// TIA Portal project "FactoryIO_Template_S7-1200_V14" (V14)
// Vorlageprojekt für das Buch mit Zielsystem S7-1200

(* hardware
DEVICE "S7-1200-Station_1"  S7-1200 Station
   slot 0: "Baugruppenträger_0"  Rack  V1.0
   slot 1: "PLC_1"  CPU 1214C DC/DC/Rly  6ES7 214-1HG40-0XB0  V4.2
   slot 3: "DQ 4x24VDC_1"  DQ4 signal board (200 kHz)  6ES7 222-1BD30-0XB0  V1.0
*)

// ===== PLC "PLC_1"  CPU 1214C DC/DC/Rly =====

VAR_GLOBAL   // PLC tag table "Standard-Variablentabelle"
   "START" AT %I0.0 : Bool;
   "STOP" AT %I0.1 : Bool;
   "M1" AT %M10.1 : Bool;
   "CONV 1" AT %Q0.0 : Bool;
   "SENSOR 1" AT %I0.2 : Bool;
   "PLAT RUN" AT %Q0.2 : Bool;
   "PLAT LIM" AT %I0.5 : Bool;
   "PLAT SPIN" AT %Q0.3 : Bool;
   "PLAT SPİND" AT %I0.3 : Bool;
   "SENSÖR 2" AT %I0.4 : Bool;
   "CONV 2" AT %Q0.1 : Bool;
   "LİFT RUN" AT %Q0.4 : Bool;
   "LİFT LİM" AT %I0.6 : Bool;
   "LİFT UP" AT %Q0.5 : Bool;
   "SENSOR 3" AT %I0.7 : Bool;
   "CONV 3" AT %Q0.6 : Bool;
   "SENSOR 4" AT %I1.0 : Bool;
   "LİFT DOWN" AT %Q0.7 : Bool;
   "LİFT 2 UP" AT %Q1.0 : Bool;
   "LİFT 2 RUN" AT %Q4.0 : Bool;
   "LİFT 2 LİM" AT %I1.1 : Bool;
   "LİFT 2 DOWN" AT %Q1.1 : Bool;
   "SENSOR 5" AT %I1.2 : Bool;
   "CONV 4" AT %Q4.1 : Bool;
   "SENSOR PM" AT %I1.3 : Bool;
END_VAR

// folder: System blocks/Program resources

DATA_BLOCK "TİMER_1"   // DB1
{ S7_Optimized_Access := 'TRUE' }
AUTHOR : Simatic
FAMILY : IEC
NAME : IEC_TMR
VERSION : 1.0
// stored: InstanceOfName IEC_TIMER
"IEC_TIMER"
BEGIN
END_DATA_BLOCK

// folder: (top level)

FUNCTION "MHJ-PLC-Lab-Function-S71200" : Void   // FC9000, SCL
{ S7_Optimized_Access := 'TRUE' }
VERSION : 0.1
   VAR_TEMP
      rdTimeReturn : Int;
      outputTime : DTL;
      SyncVal : Byte;
      forVal : Int;
      forVal_2 : Int;
      Value : Byte;
   END_VAR
   VAR CONSTANT
      CompVal : Byte := 16#34;
      Value_01 : Byte := 16#11;
      Value_01_DW : DWord := 16#A165_D992;
      Value_02_DW : DWord := 16#58BE_4401;
   END_VAR
BEGIN

   #Value:=PEEK(area := 16#82,
        dbNumber := 0,
        byteOffset := 511);
   #Value := #Value + 1;

   POKE(area := 16#82,
        dbNumber := 0,
        byteOffset := 511,
        value := #Value);

   POKE(area:=16#81,
        dbNumber:=0,
        byteOffset:=1016,
        value:=#Value_01_DW);
   POKE(area := 16#81,
        dbNumber := 0,
        byteOffset := 1020,
        value := #Value_02_DW);

   POKE(area := 16#81,
        dbNumber := 0,
        byteOffset := 511,
        value := B#16#00);

   FOR #forVal := 0 TO 120 DO
       FOR #forVal_2:=0 TO 10 DO
           #rdTimeReturn:=RD_SYS_T(#outputTime);
           #rdTimeReturn := WR_SYS_T(#outputTime);
           #rdTimeReturn := RD_SYS_T(#outputTime);
           #rdTimeReturn := WR_SYS_T(#outputTime);
       END_FOR;
       #SyncVal:= PEEK(area := 16#81,
                      dbNumber := 0,
                      byteOffset := 511);
       IF #SyncVal = #CompVal THEN
          GOTO M_1;
       END_IF;
   END_FOR;
   RETURN;

   M_1:
   POKE(area := 16#81,
        dbNumber := 0,
        byteOffset := 511,
        value := B#16#0);
END_FUNCTION

ORGANIZATION_BLOCK "Main"   // OB1, LAD, ProgramCycle
TITLE = "Main Program Sweep (Cycle)"
{ S7_Optimized_Access := 'TRUE' }
VERSION : 0.1
   VAR_INPUT
      Initial_Call : Bool;   // Initial call of this OB
      Remanence : Bool;   // =True, if remanent data are available
   END_VAR
BEGIN

REGION Network 1: Konnektierungsbaustein für PLC-Lab
   // Im Netzwerk 1 wird der Konnektierungsbaustein für PLC-Lab aufgerufen.
   // Dieser Aufruf darf nicht entfernt werden!
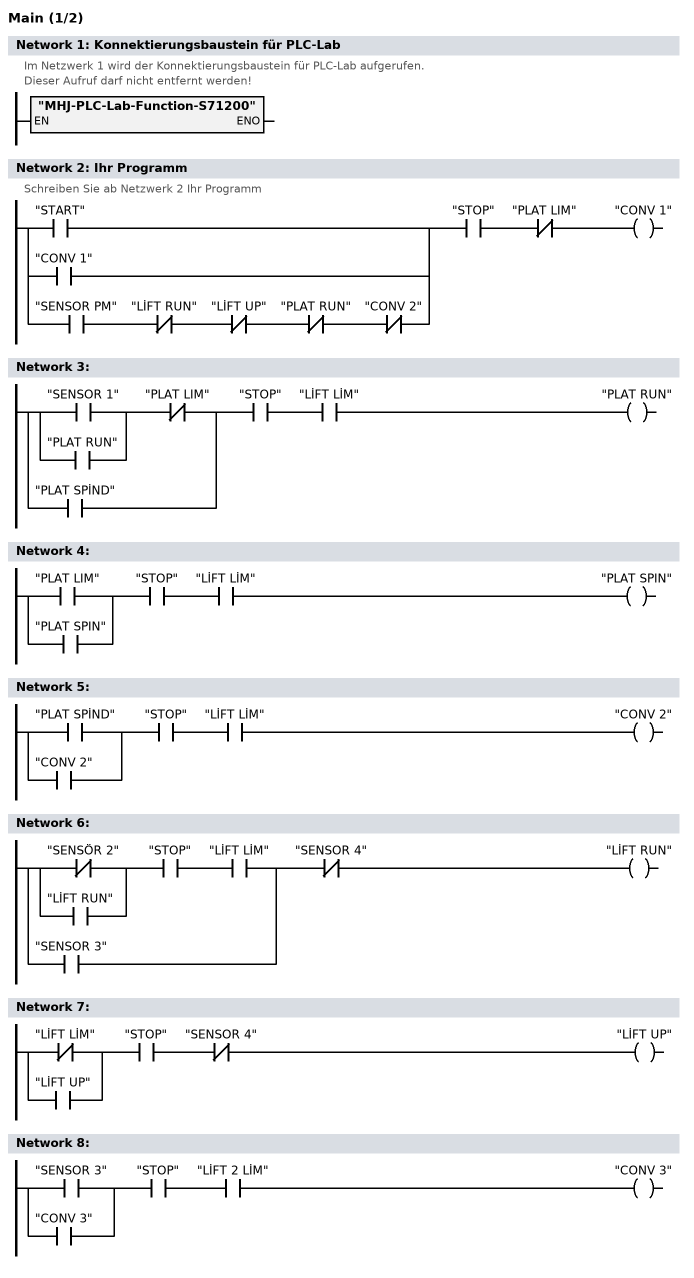
   RUNG wire#powerrail
      "MHJ-PLC-Lab-Function-S71200"()
   END_RUNG
   // the same network as SCL:
   "MHJ-PLC-Lab-Function-S71200"();
END_REGION

REGION Network 2: Ihr Programm
   // Schreiben Sie ab Netzwerk 2 Ihr Programm
   RUNG wire#powerrail
      Contact( "START" )
      wire#w1
      Contact( "STOP" )
      I_Contact( "PLAT LIM" )
      Coil( "CONV 1" )
   END_RUNG
   RUNG wire#powerrail
      Contact( "CONV 1" )
   END_RUNG wire#w1
   RUNG wire#powerrail
      Contact( "SENSOR PM" )
      I_Contact( "LİFT RUN" )
      I_Contact( "LİFT UP" )
      I_Contact( "PLAT RUN" )
      I_Contact( "CONV 2" )
   END_RUNG wire#w1
   // the same network as SCL:
   "CONV 1" := ("START" OR "CONV 1" OR ("SENSOR PM" AND NOT "LİFT RUN" AND NOT "LİFT UP" AND NOT "PLAT RUN" AND NOT "CONV 2")) AND "STOP" AND NOT "PLAT LIM";
END_REGION

REGION Network 3
   RUNG wire#powerrail
      Contact( "SENSOR 1" )
      wire#w1
      I_Contact( "PLAT LIM" )
      wire#w2
      Contact( "STOP" )
      Contact( "LİFT LİM" )
      Coil( "PLAT RUN" )
   END_RUNG
   RUNG wire#powerrail
      Contact( "PLAT RUN" )
   END_RUNG wire#w1
   RUNG wire#powerrail
      Contact( "PLAT SPİND" )
   END_RUNG wire#w2
   // the same network as SCL:
   "PLAT RUN" := ((("SENSOR 1" OR "PLAT RUN") AND NOT "PLAT LIM") OR "PLAT SPİND") AND "STOP" AND "LİFT LİM";
END_REGION

REGION Network 4
   RUNG wire#powerrail
      Contact( "PLAT LIM" )
      wire#w1
      Contact( "STOP" )
      Contact( "LİFT LİM" )
      Coil( "PLAT SPIN" )
   END_RUNG
   RUNG wire#powerrail
      Contact( "PLAT SPIN" )
   END_RUNG wire#w1
   // the same network as SCL:
   "PLAT SPIN" := ("PLAT LIM" OR "PLAT SPIN") AND "STOP" AND "LİFT LİM";
END_REGION

REGION Network 5
   RUNG wire#powerrail
      Contact( "PLAT SPİND" )
      wire#w1
      Contact( "STOP" )
      Contact( "LİFT LİM" )
      Coil( "CONV 2" )
   END_RUNG
   RUNG wire#powerrail
      Contact( "CONV 2" )
   END_RUNG wire#w1
   // the same network as SCL:
   "CONV 2" := ("PLAT SPİND" OR "CONV 2") AND "STOP" AND "LİFT LİM";
END_REGION

REGION Network 6
   RUNG wire#powerrail
      I_Contact( "SENSÖR 2" )
      wire#w1
      Contact( "STOP" )
      Contact( "LİFT LİM" )
      wire#w2
      I_Contact( "SENSOR 4" )
      Coil( "LİFT RUN" )
   END_RUNG
   RUNG wire#powerrail
      Contact( "LİFT RUN" )
   END_RUNG wire#w1
   RUNG wire#powerrail
      Contact( "SENSOR 3" )
   END_RUNG wire#w2
   // the same network as SCL:
   "LİFT RUN" := (((NOT "SENSÖR 2" OR "LİFT RUN") AND "STOP" AND "LİFT LİM") OR "SENSOR 3") AND NOT "SENSOR 4";
END_REGION

REGION Network 7
   RUNG wire#powerrail
      I_Contact( "LİFT LİM" )
      wire#w1
      Contact( "STOP" )
      I_Contact( "SENSOR 4" )
      Coil( "LİFT UP" )
   END_RUNG
   RUNG wire#powerrail
      Contact( "LİFT UP" )
   END_RUNG wire#w1
   // the same network as SCL:
   "LİFT UP" := (NOT "LİFT LİM" OR "LİFT UP") AND "STOP" AND NOT "SENSOR 4";
END_REGION

REGION Network 8
   RUNG wire#powerrail
      Contact( "SENSOR 3" )
      wire#w1
      Contact( "STOP" )
      Contact( "LİFT 2 LİM" )
      Coil( "CONV 3" )
   END_RUNG
   RUNG wire#powerrail
      Contact( "CONV 3" )
   END_RUNG wire#w1
   // the same network as SCL:
   "CONV 3" := ("SENSOR 3" OR "CONV 3") AND "STOP" AND "LİFT 2 LİM";
END_REGION

REGION Network 9
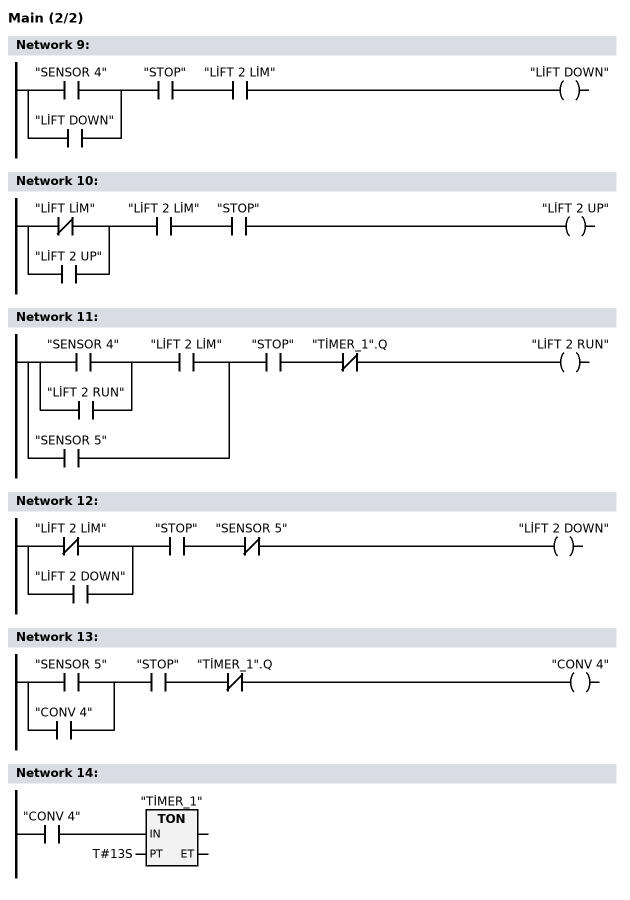
   RUNG wire#powerrail
      Contact( "SENSOR 4" )
      wire#w1
      Contact( "STOP" )
      Contact( "LİFT 2 LİM" )
      Coil( "LİFT DOWN" )
   END_RUNG
   RUNG wire#powerrail
      Contact( "LİFT DOWN" )
   END_RUNG wire#w1
   // the same network as SCL:
   "LİFT DOWN" := ("SENSOR 4" OR "LİFT DOWN") AND "STOP" AND "LİFT 2 LİM";
END_REGION

REGION Network 10
   RUNG wire#powerrail
      I_Contact( "LİFT LİM" )
      wire#w1
      Contact( "LİFT 2 LİM" )
      Contact( "STOP" )
      Coil( "LİFT 2 UP" )
   END_RUNG
   RUNG wire#powerrail
      Contact( "LİFT 2 UP" )
   END_RUNG wire#w1
   // the same network as SCL:
   "LİFT 2 UP" := (NOT "LİFT LİM" OR "LİFT 2 UP") AND "LİFT 2 LİM" AND "STOP";
END_REGION

REGION Network 11
   RUNG wire#powerrail
      Contact( "SENSOR 4" )
      wire#w1
      Contact( "LİFT 2 LİM" )
      wire#w2
      Contact( "STOP" )
      I_Contact( "TİMER_1".Q )
      Coil( "LİFT 2 RUN" )
   END_RUNG
   RUNG wire#powerrail
      Contact( "LİFT 2 RUN" )
   END_RUNG wire#w1
   RUNG wire#powerrail
      Contact( "SENSOR 5" )
   END_RUNG wire#w2
   // the same network as SCL:
   "LİFT 2 RUN" := ((("SENSOR 4" OR "LİFT 2 RUN") AND "LİFT 2 LİM") OR "SENSOR 5") AND "STOP" AND NOT "TİMER_1".Q;
END_REGION

REGION Network 12
   RUNG wire#powerrail
      I_Contact( "LİFT 2 LİM" )
      wire#w1
      Contact( "STOP" )
      I_Contact( "SENSOR 5" )
      Coil( "LİFT 2 DOWN" )
   END_RUNG
   RUNG wire#powerrail
      Contact( "LİFT 2 DOWN" )
   END_RUNG wire#w1
   // the same network as SCL:
   "LİFT 2 DOWN" := (NOT "LİFT 2 LİM" OR "LİFT 2 DOWN") AND "STOP" AND NOT "SENSOR 5";
END_REGION

REGION Network 13
   RUNG wire#powerrail
      Contact( "SENSOR 5" )
      wire#w1
      Contact( "STOP" )
      I_Contact( "TİMER_1".Q )
      Coil( "CONV 4" )
   END_RUNG
   RUNG wire#powerrail
      Contact( "CONV 4" )
   END_RUNG wire#w1
   // the same network as SCL:
   "CONV 4" := ("SENSOR 5" OR "CONV 4") AND "STOP" AND NOT "TİMER_1".Q;
END_REGION

REGION Network 14
   "TİMER_1".TON(IN := "CONV 4", PT := T#13S);
END_REGION
END_ORGANIZATION_BLOCK